// TIA Portal V18 export
TYPE "UDT_AIbasic"
// stored: IsFailsafeCompliant false
   STRUCT
      iID : DInt;   // AIs ID for monitoring
      iValue : Int;   // Int value
      rValue : Real;   // Real value
      iFilterSet : Int;   // Filter value
      rMin : Real;   // Scale Min
      rMax : Real;   // Scale Max
      wMark : String["IOmark_string_length"];   // AIs label for monitoring
   END_STRUCT;
END_TYPE
